// TIA Portal V18 export
DATA_BLOCK "NG_BOXES_DB"   // DB2911
// stored: AutoNumber false, InstanceOfName NG_BOXES, InstanceOfType FB
"NG_BOXES"
   // VAR_INPUT
   //    in_Permission_to_Open : Bool;
   // END_VAR
   // VAR_OUTPUT
   //    out_Request_to_open : Bool;
   // END_VAR
   // VAR
   //    Box_Loading { S7_SetPoint := 'True'} : "FB_NG_Box_Control";
   //    Box_Unloading { S7_SetPoint := 'True'} : "FB_NG_Box_Control";
   //    TempSensors : Array[1..15] of Bool;
   // END_VAR
BEGIN
END_DATA_BLOCK
